FUNCTION_BLOCK UT_AuxiliaryInputMapping_Type_08_DualBool_LatchedDown (* Type 8 DualBool_LatchedDown Three-position switch - latching in down position *)
  (* Standard: ISO 11783-6; Classification: AUX – ISO 11783-6; Function: All Inputs; Type: UT according to ISO 11783-6; Description: Copyright (c) 2018, 2023 Jose Cabral, HR Agrartechnik GmbH This program and the accompanying materials are made available under the terms of the Eclipse Public License 2.0 which is available at https://www.eclipse.org/legal/epl-2.0/ SPDX-License-Identifier: EPL-2.0 - Type 8 DualBool_LatchedDown Three-position switch - latching in down position Applicable AUX-N only * Maps to IX *)
  (* Version 1.0, 2018-12-05, Jose Cabral *)
  (* Version 1.1, 2022-08-04, Franz Höpfinger, HR Agrartechnik GmbH *)
  (* Version 1.2, 2023-01-05, Franz Höpfinger, HR Agrartechnik GmbH *)
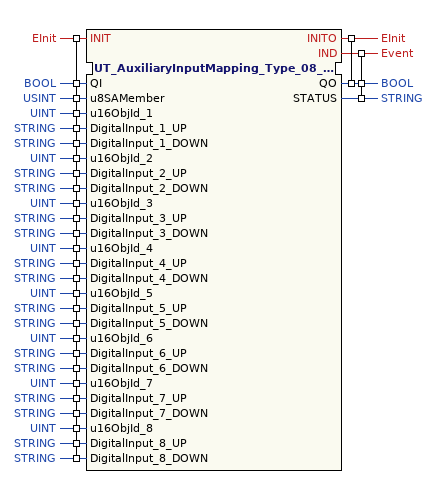
  EVENT_INPUT
    INIT : EInit WITH QI, u8SAMember, u16ObjId_1, DigitalInput_1_UP, DigitalInput_1_DOWN, u16ObjId_2, DigitalInput_2_UP, DigitalInput_2_DOWN, u16ObjId_3, DigitalInput_3_UP, DigitalInput_3_DOWN, u16ObjId_4, DigitalInput_4_UP, DigitalInput_4_DOWN, u16ObjId_5, DigitalInput_5_UP, DigitalInput_5_DOWN, u16ObjId_6, DigitalInput_6_UP, DigitalInput_6_DOWN, u16ObjId_7, DigitalInput_7_UP, DigitalInput_7_DOWN, u16ObjId_8, DigitalInput_8_UP, DigitalInput_8_DOWN; (* Service Initialization *)
  END_EVENT
  EVENT_OUTPUT
    INITO : EInit WITH QO; (* Initialization Confirm *)
    IND WITH QO, STATUS; (* Indication from Resource *)
  END_EVENT
  VAR_INPUT
    QI : BOOL; (* Event Input Qualifier *)
    u8SAMember : USINT := isobus::GLOBAL; (* Dummy !, set to GLOBAL if in doubt. OFF deactivates FB. *)
    u16ObjId_1 : UINT; (* Object ID of Input 1 *)
    DigitalInput_1_UP : STRING; (* Identifier for Input 1 UP *)
    DigitalInput_1_DOWN : STRING; (* Identifier for Input 1 DOWN *)
    u16ObjId_2 : UINT; (* Object ID of Input 2 *)
    DigitalInput_2_UP : STRING; (* Identifier for Input 2 UP *)
    DigitalInput_2_DOWN : STRING; (* Identifier for Input 2 DOWN *)
    u16ObjId_3 : UINT; (* Object ID of Input 3 *)
    DigitalInput_3_UP : STRING; (* Identifier for Input 3 UP *)
    DigitalInput_3_DOWN : STRING; (* Identifier for Input 3 DOWN *)
    u16ObjId_4 : UINT; (* Object ID of Input 4 *)
    DigitalInput_4_UP : STRING; (* Identifier for Input 4 UP *)
    DigitalInput_4_DOWN : STRING; (* Identifier for Input 4 DOWN *)
    u16ObjId_5 : UINT; (* Object ID of Input 5 *)
    DigitalInput_5_UP : STRING; (* Identifier for Input 5 UP *)
    DigitalInput_5_DOWN : STRING; (* Identifier for Input 5 DOWN *)
    u16ObjId_6 : UINT; (* Object ID of Input 6 *)
    DigitalInput_6_UP : STRING; (* Identifier for Input 6 UP *)
    DigitalInput_6_DOWN : STRING; (* Identifier for Input 6 DOWN *)
    u16ObjId_7 : UINT; (* Object ID of Input 7 *)
    DigitalInput_7_UP : STRING; (* Identifier for Input 7 UP *)
    DigitalInput_7_DOWN : STRING; (* Identifier for Input 7 DOWN *)
    u16ObjId_8 : UINT; (* Object ID of Input 8 *)
    DigitalInput_8_UP : STRING; (* Identifier for Input 8 UP *)
    DigitalInput_8_DOWN : STRING; (* Identifier for Input 8 DOWN *)
  END_VAR
  VAR_OUTPUT
    QO : BOOL; (* Event Output Qualifier *)
    STATUS : STRING; (* Service Status *)
  END_VAR
END_FUNCTION_BLOCK
